Universal Robots PolyScope program: cobot.urp

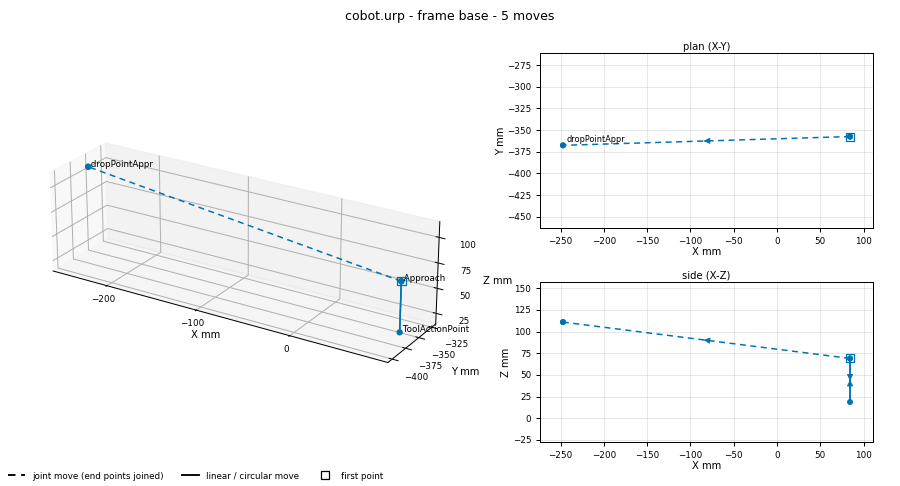
[picture p0: tool path of cobot.urp in frame base, 5 of 5 moves have a stored position in this frame; points joined in program order, loops and branches not executed]
Program cobot (installation=default directory=/programs/usbdisk_0 createdIn=5.12.1.1101497 lastSavedIn=5.12.1.1101497 robotSerialNumber=20225300640)
Calibrated DH parameters: a=[-0.000125, -0.240482, -0.204397, 0.000169, -0.000135, 0]; d=[0.152056, 4.760815, 12.138494, -16.768367, 0.085457, 0.092357]; alpha=[1.570863, 0.008548, 0.003635, 1.571424, -1.571918, 0]; deltaTheta=[0, 0.167622, 0.124346, -0.291972, 0.000034, 0]
Robot Program (runOnlyOnce=false)
  SafeHome (positionOptionType=SPEED_AND_ACCELERATION speed=1.047198 acceleration=1.396263 nextMotionTime=2)
  Set DigitalOutput pin=digital_out[2]; digitalValue=0
  Set DigitalOutput pin=digital_out[1]; digitalValue=1
  URCap Palletizing (polyscope-pallet-impl, Universal Robots) dataModel(palletFeature=Base, isPalletizing=true, rememberTraversal=false, Variable(key=name, variable(name=Pallet_1)), Variable(key=layerNumberVariable, variable(name=Pallet_1_lno, initializeExpression=1)), Variable(key=layerCountingVariable, variable(name=Pallet_1_lct, initializeExpression=1)), Variable(key=handleSeparatorVariable, variable(name=Pallet_1_sep, initializeExpression=False)), Variable(key=totalCountVariable, variable(name=Pallet_1_tct, initializeExpression=1)), Variable(key=referencePoint, variable(featureName=referencePoint)), Variable(key=separatorPoint, variable(featureName=separatorPoint)), Length(key=objectHeight value=0.015 unit=M), Variable(key=globalCountingVariable, variable(name=Pallet_1_cnt_2, initializeExpression=1))); state(isChildrenLocked=true)
    URCap Patterns (polyscope-pallet-impl, Universal Robots) state(isChildrenLocked=true)
      URCap Pattern (polyscope-pallet-impl, Universal Robots) dataModel(UUID=ff210ff5-9ef1-4973-bc2b-4b7444e62114, patternType=IRREGULAR, Variable(key=nameVariable, variable(name=Irreg_Pattern_1))); state(isChildrenLocked=true)
        URCap Item (polyscope-pallet-impl, Universal Robots) dataModel(UUID=946cba2f-218f-425b-a796-11d9354ba379, patternType=IRREGULAR, index=0, calibrationDeltaTheta=[-4.022425301349053E-7, 0.1676224840059082, 0.12434612800300923, -0.29197201232783093, 3.427063592260221E-5, -2.1055269264214083E-9], calibrationA=[-1.2536318386722594E-4, -0.24048217598078755, -0.20439712606180582, 1.6856812341359539E-4, -1.3512489031768148E-4, 0.0], calibrationD=[0.1520559623222255, 4.760815016703785, 12.138493934059257, -16.768366633975226, 0.08545691164632878, 0.09235657960129308], calibrationAlpha=[1.570862629498801, 0.008547662301921876, 0.0036353825850200293, 1.5714242532258311, -1.5719182813352055, 0.0], calibrationJointChecksum=[-1442419114, -1443167645, -1459096000, -1465254611, -1461595521, -1465327861], calibrationStatus=2, calibrationValidChecksum=true, baseToFeature=[0.0, 0.0, 0.0, 0.0, 0.0, 0.0], TCPOffset=[9.97898322563362E-6, 1.3955372514251607E-5, 0.14500591279719433, -4.958366891809747E-5, 5.261404997077385E-6, 2.988673267554275E-5], Variable(key=variable, variable(name=Item_1)), JointPositions(key=jointpositions, JointPosition(key=[1], Angle(key=pos value=1.414477 unit=RAD)), JointPosition(key=[2], Angle(key=pos value=-1.236849 unit=RAD)), JointPosition(key=[3], Angle(key=pos value=1.884528 unit=RAD)), JointPosition(key=[4], Angle(key=pos value=-2.234845 unit=RAD)), JointPosition(key=[5], Angle(key=pos value=-1.523196 unit=RAD)), JointPosition(key=[6], Angle(key=pos value=-0.155582 unit=RAD))))
        URCap Item (polyscope-pallet-impl, Universal Robots) dataModel(UUID=5718a253-88ac-41d8-8b33-e7b171991ae4, patternType=IRREGULAR, index=1, calibrationDeltaTheta=[-4.022425301349053E-7, 0.1676224840059082, 0.12434612800300923, -0.29197201232783093, 3.427063592260221E-5, -2.1055269264214083E-9], calibrationA=[-1.2536318386722594E-4, -0.24048217598078755, -0.20439712606180582, 1.6856812341359539E-4, -1.3512489031768148E-4, 0.0], calibrationD=[0.1520559623222255, 4.760815016703785, 12.138493934059257, -16.768366633975226, 0.08545691164632878, 0.09235657960129308], calibrationAlpha=[1.570862629498801, 0.008547662301921876, 0.0036353825850200293, 1.5714242532258311, -1.5719182813352055, 0.0], calibrationJointChecksum=[-1442419114, -1443167645, -1459096000, -1465254611, -1461595521, -1465327861], calibrationStatus=2, calibrationValidChecksum=true, baseToFeature=[0.0, 0.0, 0.0, 0.0, 0.0, 0.0], TCPOffset=[-2.206079688518714E-5, -7.55269417079818E-6, 0.14499230985935901, 5.326253605900404E-5, 4.831116813240864E-6, -7.363332137093319E-5], Variable(key=variable, variable(name=Item_2)), JointPositions(key=jointpositions, JointPosition(key=[1], Angle(key=pos value=1.199839 unit=RAD)), JointPosition(key=[2], Angle(key=pos value=-1.253531 unit=RAD)), JointPosition(key=[3], Angle(key=pos value=1.891806 unit=RAD)), JointPosition(key=[4], Angle(key=pos value=-2.178204 unit=RAD)), JointPosition(key=[5], Angle(key=pos value=-1.566813 unit=RAD)), JointPosition(key=[6], Angle(key=pos value=-0.327061 unit=RAD))))
        URCap Item (polyscope-pallet-impl, Universal Robots) dataModel(UUID=d95725a4-8d9a-4d6e-ad82-e2394f9d7de1, patternType=IRREGULAR, index=2, calibrationDeltaTheta=[-4.022425301349053E-7, 0.1676224840059082, 0.12434612800300923, -0.29197201232783093, 3.427063592260221E-5, -2.1055269264214083E-9], calibrationA=[-1.2536318386722594E-4, -0.24048217598078755, -0.20439712606180582, 1.6856812341359539E-4, -1.3512489031768148E-4, 0.0], calibrationD=[0.1520559623222255, 4.760815016703785, 12.138493934059257, -16.768366633975226, 0.08545691164632878, 0.09235657960129308], calibrationAlpha=[1.570862629498801, 0.008547662301921876, 0.0036353825850200293, 1.5714242532258311, -1.5719182813352055, 0.0], calibrationJointChecksum=[-1442419114, -1443167645, -1459096000, -1465254611, -1461595521, -1465327861], calibrationStatus=2, calibrationValidChecksum=true, baseToFeature=[0.0, 0.0, 0.0, 0.0, 0.0, 0.0], TCPOffset=[4.9270793688604986E-6, -8.692108637964324E-6, 0.1449907283398865, 3.4176372793594984E-5, 2.7932800995310264E-5, -1.4703926023480856E-5], Variable(key=variable, variable(name=Item_3)), JointPositions(key=jointpositions, JointPosition(key=[1], Angle(key=pos value=0.925998 unit=RAD)), JointPosition(key=[2], Angle(key=pos value=-1.230368 unit=RAD)), JointPosition(key=[3], Angle(key=pos value=1.868108 unit=RAD)), JointPosition(key=[4], Angle(key=pos value=-2.195625 unit=RAD)), JointPosition(key=[5], Angle(key=pos value=-1.541486 unit=RAD)), JointPosition(key=[6], Angle(key=pos value=-0.587612 unit=RAD))))
        URCap Item (polyscope-pallet-impl, Universal Robots) dataModel(UUID=7a657981-3bac-44e9-81e2-025659327ee9, patternType=IRREGULAR, index=3, calibrationDeltaTheta=[-4.022425301349053E-7, 0.1676224840059082, 0.12434612800300923, -0.29197201232783093, 3.427063592260221E-5, -2.1055269264214083E-9], calibrationA=[-1.2536318386722594E-4, -0.24048217598078755, -0.20439712606180582, 1.6856812341359539E-4, -1.3512489031768148E-4, 0.0], calibrationD=[0.1520559623222255, 4.760815016703785, 12.138493934059257, -16.768366633975226, 0.08545691164632878, 0.09235657960129308], calibrationAlpha=[1.570862629498801, 0.008547662301921876, 0.0036353825850200293, 1.5714242532258311, -1.5719182813352055, 0.0], calibrationJointChecksum=[-1442419114, -1443167645, -1459096000, -1465254611, -1461595521, -1465327861], calibrationStatus=2, calibrationValidChecksum=true, baseToFeature=[0.0, 0.0, 0.0, 0.0, 0.0, 0.0], TCPOffset=[7.863421526699277E-6, 2.2464432848368077E-6, 0.14497936571115647, -2.592652631981696E-5, 3.663766306514172E-5, 3.644127181374989E-5], Variable(key=variable, variable(name=Item_4)), JointPositions(key=jointpositions, JointPosition(key=[1], Angle(key=pos value=1.105066 unit=RAD)), JointPosition(key=[2], Angle(key=pos value=-0.858452 unit=RAD)), JointPosition(key=[3], Angle(key=pos value=1.240504 unit=RAD)), JointPosition(key=[4], Angle(key=pos value=-1.94688 unit=RAD)), JointPosition(key=[5], Angle(key=pos value=-1.522029 unit=RAD)), JointPosition(key=[6], Angle(key=pos value=-2.176443 unit=RAD))))
        URCap Item (polyscope-pallet-impl, Universal Robots) dataModel(UUID=dddd6f06-cf05-43fa-94bd-864ad3a1f586, patternType=IRREGULAR, index=4, calibrationDeltaTheta=[-4.022425301349053E-7, 0.1676224840059082, 0.12434612800300923, -0.29197201232783093, 3.427063592260221E-5, -2.1055269264214083E-9], calibrationA=[-1.2536318386722594E-4, -0.24048217598078755, -0.20439712606180582, 1.6856812341359539E-4, -1.3512489031768148E-4, 0.0], calibrationD=[0.1520559623222255, 4.760815016703785, 12.138493934059257, -16.768366633975226, 0.08545691164632878, 0.09235657960129308], calibrationAlpha=[1.570862629498801, 0.008547662301921876, 0.0036353825850200293, 1.5714242532258311, -1.5719182813352055, 0.0], calibrationJointChecksum=[-1442419114, -1443167645, -1459096000, -1465254611, -1461595521, -1465327861], calibrationStatus=2, calibrationValidChecksum=true, baseToFeature=[0.0, 0.0, 0.0, 0.0, 0.0, 0.0], TCPOffset=[2.337896764625924E-6, -7.467706634525784E-7, 0.14501093329201414, -4.5951162972875905E-5, -6.811232132057431E-6, -1.6050896851225674E-5], Variable(key=variable, variable(name=Item_5)), JointPositions(key=jointpositions, JointPosition(key=[1], Angle(key=pos value=1.419045 unit=RAD)), JointPosition(key=[2], Angle(key=pos value=-0.859412 unit=RAD)), JointPosition(key=[3], Angle(key=pos value=1.252348 unit=RAD)), JointPosition(key=[4], Angle(key=pos value=-1.982103 unit=RAD)), JointPosition(key=[5], Angle(key=pos value=-1.552526 unit=RAD)), JointPosition(key=[6], Angle(key=pos value=-1.760095 unit=RAD))))
    URCap Layers (polyscope-pallet-impl, Universal Robots) dataModel(separators=[false], selectedPatterns=[ff210ff5-9ef1-4973-bc2b-4b7444e62114])
    URCap At Each Item (polyscope-pallet-impl, Universal Robots) dataModel(selectedPattern=ff210ff5-9ef1-4973-bc2b-4b7444e62114, selectedPosition=946cba2f-218f-425b-a796-11d9354ba379, Approach_calibrationDeltaTheta=[-4.022425301349053E-7, 0.1676224840059082, 0.12434612800300923, -0.29197201232783093, 3.427063592260221E-5, -2.1055269264214083E-9], Approach_calibrationA=[-1.2536318386722594E-4, -0.24048217598078755, -0.20439712606180582, 1.6856812341359539E-4, -1.3512489031768148E-4, 0.0], Approach_calibrationD=[0.1520559623222255, 4.760815016703785, 12.138493934059257, -16.768366633975226, 0.08545691164632878, 0.09235657960129308], Approach_calibrationAlpha=[1.570862629498801, 0.008547662301921876, 0.0036353825850200293, 1.5714242532258311, -1.5719182813352055, 0.0], Approach_calibrationJointChecksum=[-1442419114, -1443167645, -1459096000, -1465254611, -1461595521, -1465327861], Approach_calibrationStatus=2, Approach_calibrationValidChecksum=true, Approach_baseToFeature=[0.0, 0.0, 0.0, 0.0, 0.0, 0.0], Approach_TCPOffset=[-1.7725585822608858E-6, -4.664080850091956E-6, 0.1449886023174107, 4.226698510504133E-5, 1.936632576761414E-5, 7.716305606405693E-6], Exit_calibrationDeltaTheta=[-4.022425301349053E-7, 0.1676224840059082, 0.12434612800300923, -0.29197201232783093, 3.427063592260221E-5, -2.1055269264214083E-9], Exit_calibrationA=[-1.2536318386722594E-4, -0.24048217598078755, -0.20439712606180582, 1.6856812341359539E-4, -1.3512489031768148E-4, 0.0], Exit_calibrationD=[0.1520559623222255, 4.760815016703785, 12.138493934059257, -16.768366633975226, 0.08545691164632878, 0.09235657960129308], Exit_calibrationAlpha=[1.570862629498801, 0.008547662301921876, 0.0036353825850200293, 1.5714242532258311, -1.5719182813352055, 0.0], Exit_calibrationJointChecksum=[-1442419114, -1443167645, -1459096000, -1465254611, -1461595521, -1465327861], Exit_calibrationStatus=2, Exit_calibrationValidChecksum=true, Exit_baseToFeature=[0.0, 0.0, 0.0, 0.0, 0.0, 0.0], Exit_TCPOffset=[-1.2076336013633338E-5, 1.0908497542150286E-5, 0.14500763303586645, -2.471728327552712E-5, -1.5762579468986066E-5, -2.3791396451331094E-5], currentWizardState=SHOW_DONE, Pose(key=refBaseToFeature, Position(key=posePosition, Length(key=X value=0 unit=M), Length(key=Y value=0 unit=M), Length(key=Z value=0 unit=M)), Rotation(key=poseRotation, Angle(key=RX value=0 unit=RAD), Angle(key=RY value=0 unit=RAD), Angle(key=RZ value=0 unit=RAD))), Pose(key=refPose, Position(key=posePosition, Length(key=X value=0.084293 unit=M), Length(key=Y value=-0.357458 unit=M), Length(key=Z value=0.018636 unit=M)), Rotation(key=poseRotation, Angle(key=RX value=0.008459 unit=RAD), Angle(key=RY value=3.102998 unit=RAD), Angle(key=RZ value=-0.033429 unit=RAD))), JointPositions(key=Approach_jointpositions, JointPosition(key=[1], Angle(key=pos value=1.414806 unit=RAD)), JointPosition(key=[2], Angle(key=pos value=-1.347738 unit=RAD)), JointPosition(key=[3], Angle(key=pos value=1.75337 unit=RAD)), JointPosition(key=[4], Angle(key=pos value=-1.992688 unit=RAD)), JointPosition(key=[5], Angle(key=pos value=-1.523456 unit=RAD)), JointPosition(key=[6], Angle(key=pos value=-0.15626 unit=RAD))), JointPositions(key=Exit_jointpositions, JointPosition(key=[1], Angle(key=pos value=1.414757 unit=RAD)), JointPosition(key=[2], Angle(key=pos value=-1.347719 unit=RAD)), JointPosition(key=[3], Angle(key=pos value=1.753354 unit=RAD)), JointPosition(key=[4], Angle(key=pos value=-1.992702 unit=RAD)), JointPosition(key=[5], Angle(key=pos value=-1.523383 unit=RAD)), JointPosition(key=[6], Angle(key=pos value=-0.156305 unit=RAD))))
      URCap Generated Movements (polyscope-pallet-impl, Universal Robots) state(isChildrenLocked=true)
        MoveJ speed 60 deg/s, acceleration 80 deg/s^2 (useActiveTCP=true) feature=referencePoint
          Waypoint Approach: TCP in base x=84.287 y=-357.451 z=69.012 mm, rx=0.0085 ry=3.1031 rz=-0.0334 rad; joints [82.016, -52.576, 112.58, -150.986, -87.246, -7.809] deg; TCP offset x=0 y=0 z=0 mm, rx=0 ry=0 rz=0 rad; feature pose in base x=84.293 y=-357.458 z=18.636 mm, rx=0.0085 ry=3.103 rz=-0.0334 rad
        MoveL speed 250 mm/s, acceleration 1200 mm/s^2 (useActiveTCP=true) feature(featureName=referencePoint)
          Waypoint ToolActionPoint: TCP in base x=84.293 y=-357.458 z=18.636 mm, rx=0.0085 ry=3.103 rz=-0.0334 rad; joints [81.997, -40.948, 111.558, -161.594, -87.221, -7.745] deg; TCP offset x=0 y=0 z=0 mm, rx=0 ry=0 rz=0 rad
        Folder Tool action
          URCap Vacuum (Robotiq_Grippers, Robotiq Inc.) dataModel(Vacuum.Command.ReleaseOptionWaitObjectRelease=true, Vacuum.Command.GripOptionWaitForObjectDetected=false, Vacuum.Command.Action=0, Vacuum.Command.GripMode=Manual, Vacuum.Command.PumpAutoCloseDelayInMilliseconds=3000, Vacuum.Command.ShutOffDistance=5.0)
          Wait Sleep waitTime=0.5
          URCap Grip Check (Robotiq_Grippers, Robotiq Inc.) dataModel(DimensionKey=100.0, DimensionDimensionPositiveGapKey=5.0, DimensionNegativeGapKey=5.0, GripperIdKey=1, ModelDefinedKey=true, ObjectDetectedKey=false, DimensionValidationKey=false); state(isChildrenLocked=true)
            URCap If (Robotiq_Grippers, Robotiq Inc.)
              Set IncrementVariable installationVariable=Pallet_1_cnt_1
              Set DigitalOutput pin=digital_out[2]; digitalValue=1
        MoveL speed 250 mm/s, acceleration 1200 mm/s^2 (useActiveTCP=true) feature(featureName=referencePoint)
          Waypoint Exit_1: TCP in base x=84.297 y=-357.449 z=68.993 mm, rx=0.0085 ry=3.103 rz=-0.0334 rad; joints [82.016, -52.572, 112.58, -150.986, -87.241, -7.811] deg; TCP offset x=0 y=0 z=0 mm, rx=0 ry=0 rz=0 rad
      MoveJ speed 60 deg/s, acceleration 80 deg/s^2 (useActiveTCP=true) feature=Base
        Waypoint dropPointAppr: TCP in base x=-247.157 y=-367.587 z=110.973 mm, rx=2.2331 ry=2.1714 rz=-0.13 rad; joints [38.055, -64.528, 72.748, -102.879, -87.617, 39.428] deg; TCP offset x=0 y=0 z=145 mm, rx=0 ry=0 rz=0 rad
      MoveL speed 250 mm/s, acceleration 1200 mm/s^2 (useActiveTCP=true) feature=Base
        MoveDirectionNode (selectedDirection=ZMinus toolParams=0.05, 1.2)
          Until TOOL_CONTACT_DETECTION (allowActions=true retraction=0 decelerationAcceleration=1.2 decelerationAngularAcceleration=34.906585)
            URCap Vacuum (Robotiq_Grippers, Robotiq Inc.) dataModel(Vacuum.Command.GripOptionWaitForObjectDetected=false, Vacuum.Command.Action=1, Vacuum.Command.PumpAutoCloseDelayInMilliseconds=3000, Vacuum.Command.ShutOffDistance=5.0)
      MoveJ speed 60 deg/s, acceleration 80 deg/s^2 (useActiveTCP=true) feature=Base
        Waypoint dropPointAppr: TCP in base x=-247.157 y=-367.587 z=110.973 mm, rx=2.2331 ry=2.1714 rz=-0.13 rad; joints [38.055, -64.528, 72.748, -102.879, -87.617, 39.428] deg
